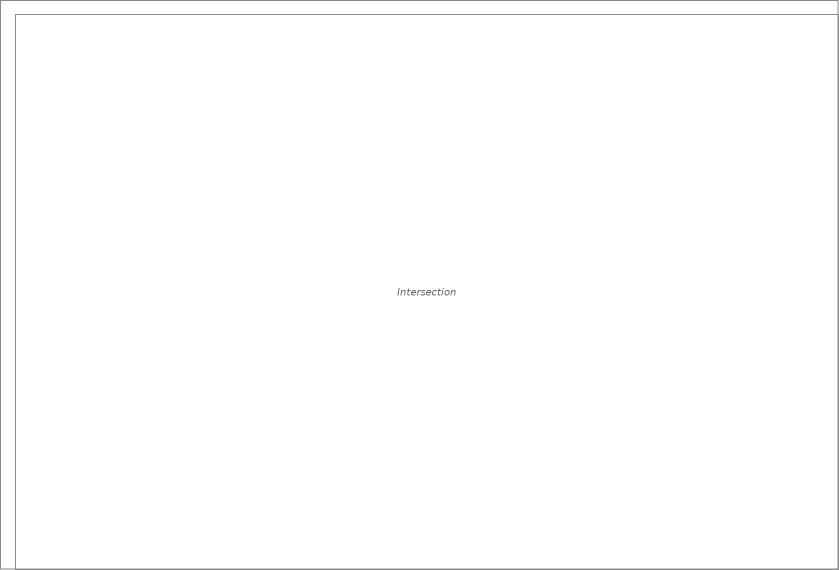
VISUALIZATION MainVisualization  // 839x570
    TabControl (15,14 824x556)
        shows Intersection()
        shows Workflow()
        [0]: TabTitle=Intersection
        [1]: TabTitle=Workflow
END_VISUALIZATION

(* stored: Version 1.1.0.1
   Visu MainVisualization: Id {5eda6eb3-8541-43ab-8edd-578aa1e092e4} *)
